// TIA Portal V20 export
DATA_BLOCK "DB_Machineshutdown_UPS"   // DB461
// stored: AutoNumber false, InstanceOfName FB_Machineshutdown_UPS, InstanceOfType FB
"FB_Machineshutdown_UPS"
   // VAR
   //    sTimeOutShutDown { S7_SetPoint := 'True'} : TON_TIME;
   //    sTimeOutAlarmUPS { S7_SetPoint := 'True'} : TON_TIME;
   //    sTimeOutShutDownPC { S7_SetPoint := 'True'} : TON_TIME;
   //    sShutDownDelayPC { S7_SetPoint := 'True'} : TON_TIME;
   //    sShutDownAspiration : Bool;
   //    sShutDownPower : Bool;
   //    sShutDownPCRequest : Int;
   //    sShutDownPCResponse : Int;
   // END_VAR
BEGIN
END_DATA_BLOCK
